BCV_222_CTRL(OL := GVL.S8605[s8605_Mapping.SV_222].PDO.DI2, CL := GVL.S8605[s8605_Mapping.SV_222].PDO.DI1, LOCKOUT := False, Online := GVL.S8605[s8605_Mapping.SV_222].PDO.Namur.eNamur<>Burkert.eNamur107.Offline, Interlock := False, BCV := GVL.BCV[BCV_Mapping.BCV_222], Output => GVL.S8605[s8605_Mapping.SV_222].PDO.DO1);

BCV_223_CTRL(OL := GVL.S8605[s8605_Mapping.SV_223].PDO.DI2, CL := GVL.S8605[s8605_Mapping.SV_223].PDO.DI1, LOCKOUT := False, Online := GVL.S8605[s8605_Mapping.SV_223].PDO.Namur.eNamur<>Burkert.eNamur107.Offline, Interlock := False, BCV := GVL.BCV[BCV_Mapping.BCV_223], Output => GVL.S8605[s8605_Mapping.SV_223].PDO.DO1);
END_PROGRAM
